SUBAPPLICATION Uebung_039a (* Spiegelabfolge V2 mit Schrittkette *)
  (* Standard: 61499-2; Description: Spiegelabfolge V2 mit Schrittkette geeignet für hydraulisches Ringsystem 3/2 Wege Ventile  (z.B. Claas) oder pneumatische 5/2 Wege Ventile *)
  (* Version 1.0, 2023-10-23, franz *)
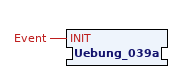
  EVENT_INPUT
    INIT;
  END_EVENT
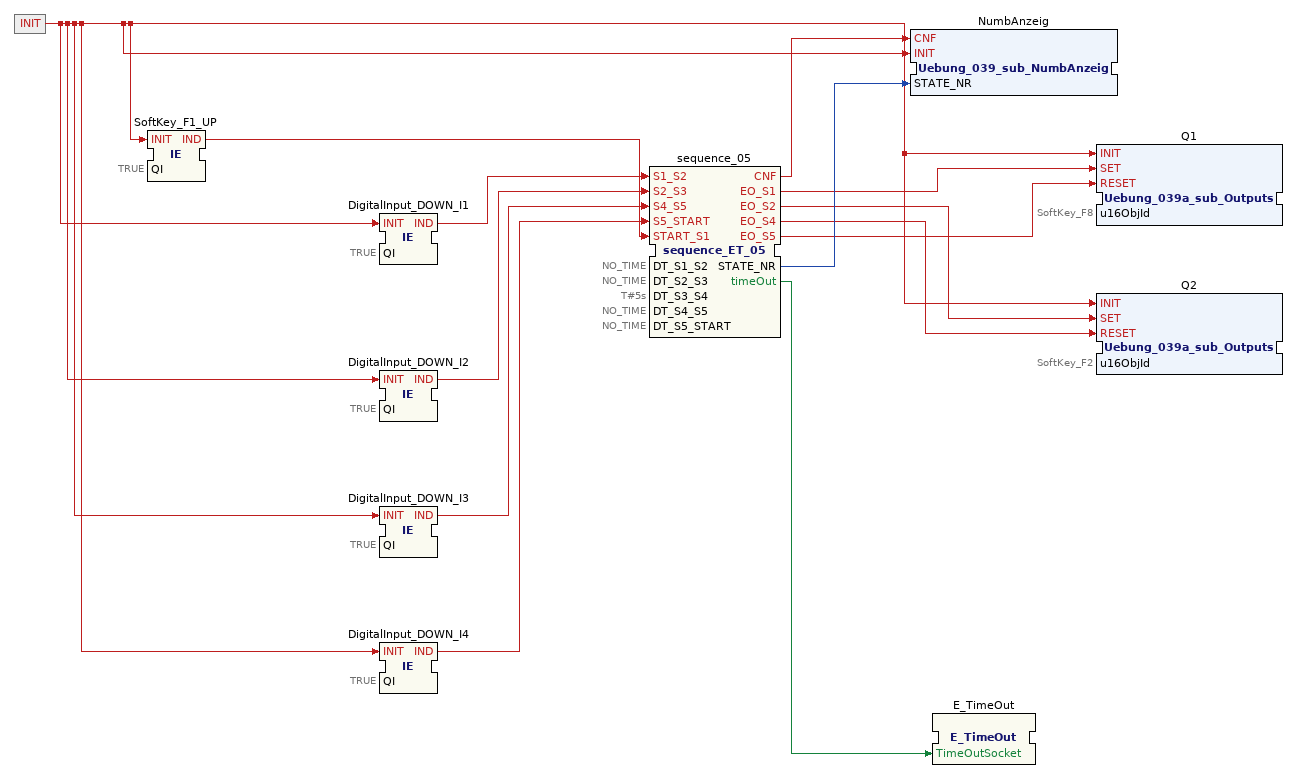
  FBS
    E_TimeOut : E_TimeOut;
    DigitalInput_DOWN_I1 : IE(QI := TRUE);
    DigitalInput_DOWN_I2 : IE(QI := TRUE);
    DigitalInput_DOWN_I3 : IE(QI := TRUE);
    DigitalInput_DOWN_I4 : IE(QI := TRUE);
    sequence_05 : sequence_ET_05(DT_S1_S2 := NO_TIME, DT_S2_S3 := NO_TIME, DT_S3_S4 := T#5s, DT_S4_S5 := NO_TIME, DT_S5_START := NO_TIME);
    SoftKey_F1_UP : IE(QI := TRUE);
  END_FBS
  SUBAPPS
    NumbAnzeig : Uebung_039_sub_NumbAnzeig;
    Q1 : Uebung_039a_sub_Outputs(u16ObjId := SoftKey_F8);
    Q2 : Uebung_039a_sub_Outputs(u16ObjId := SoftKey_F2);
  END_SUBAPPS
  EVENT_CONNECTIONS
    INIT TO DigitalInput_DOWN_I1.INIT;
    INIT TO DigitalInput_DOWN_I2.INIT;
    INIT TO DigitalInput_DOWN_I3.INIT;
    INIT TO DigitalInput_DOWN_I4.INIT;
    DigitalInput_DOWN_I1.IND TO sequence_05.S1_S2;
    DigitalInput_DOWN_I2.IND TO sequence_05.S2_S3;
    DigitalInput_DOWN_I3.IND TO sequence_05.S4_S5;
    DigitalInput_DOWN_I4.IND TO sequence_05.S5_START;
    sequence_05.CNF TO NumbAnzeig.CNF;
    INIT TO NumbAnzeig.INIT;
    INIT TO SoftKey_F1_UP.INIT;
    SoftKey_F1_UP.IND TO sequence_05.START_S1;
    INIT TO Q1.INIT;
    INIT TO Q2.INIT;
    sequence_05.EO_S1 TO Q1.SET;
    sequence_05.EO_S2 TO Q2.SET;
    sequence_05.EO_S4 TO Q2.RESET;
    sequence_05.EO_S5 TO Q1.RESET;
  END_CONNECTIONS
  DATA_CONNECTIONS
    sequence_05.STATE_NR TO NumbAnzeig.STATE_NR;
  END_CONNECTIONS
  ADAPTER_CONNECTIONS
    sequence_05.timeOut TO E_TimeOut.TimeOutSocket;
  END_CONNECTIONS
END_SUBAPPLICATION
